// TIA Portal V16 export
// export: Created 2021-11-12T13:31:53.2296923Z, ExportSetting WithDefaults, DisplayName Totally Integrated Automation Portal, DisplayVersion V16 Update 3, DisplayName TIA Portal Version Control Interface, DisplayVersion V16 Update 2, DisplayName TIA Portal Openness, DisplayVersion V16 Update 3, DisplayName SINAMICS Startdrive Advanced, DisplayVersion V16 Update 5, DisplayName SINAMICS Startdrive G130, G150, S120, S150, SINAMICS MV, S210, DisplayVersion V16 Update 5, DisplayName SINAMICS Startdrive G110M, G120, G120C, G120D, G120P, G115D, DisplayVersion V16 Update 5, DisplayName STEP 7 Professional, DisplayVersion V16 Update 3, DisplayName STEP 7 Safety, DisplayVersion V16, DisplayName WinCC UA Professional, DisplayVersion V16 Update 3
DATA_BLOCK "STATUS_000+UH10"   // DB60
{ S7_Optimized_Access := 'TRUE' }
VERSION : 0.1
// stored: AutoNumber true, DBAccessibleFromOPCUA true, IsOnlyStoredInLoadMemory false, IsRetainMemResEnabled false, IsWriteProtectedInAS false, MemoryReserve 100
   VAR
      xxxxx___BinarySensors___xxxxx : Byte;
      xxxxx___BinaryOthers___xxxxx : Byte;
      EC01_3 : Bool;   // Chlazení rozvaděče Vstupní filtr Centrální pult UH10 OK
      FC21_14 : Bool;   // Napájení 230V Centrální pult UH10 UPS OK
      FC22_14 : Bool;   // Napájení 230V Centrální pult UH10 Zásuvky OK
      FB02_14 : Bool;   // Napájení 230V Centrální pult UH10 Servisní zásuvky OK
      SF02_14 : Bool;   // Start automat
      SF03_14 : Bool;   // Nulování poruchy
      SF04_14 : Bool;   // Reset bezpečnostního okruhu
      "I452.7" : Bool;   // Rezerva res10
      SF06_14 : Bool;   // Osvětlení kamer Zóna 1
      SF07_14 : Bool;   // Osvětlení kamer Zóna 2
      SF08_14 : Bool;   // Osvětlení kamer Zóna 3
      SF09_14 : Bool;   // Osvětlení kamer Zóna 4
      "I453.4" : Bool;   // Rezerva res15
      "I453.5" : Bool;   // Rezerva res16
      "I453.7" : Bool;   // Rezerva res4
      SF14_22 : Bool;   // Blokování pásu v peci 1
      SF15_22 : Bool;   // Blokování pásu v peci 2
      SF16_22 : Bool;   // Blokování pásu v peci 3
      SF17_22 : Bool;   // Blokování dopravníku chlazení 1
      SF18_22 : Bool;   // Blokování pásu v peci 4
      SF19_22 : Bool;   // Blokování dopravníku chlazení 2
      SF20_22 : Bool;   // Blokování pásu v peci 5
      SF21_22 : Bool;   // Blokování dopravníku chlazení 3
      SF22_14 : Bool;   // Přemostění Safe move 2R1, 2R2
      "I455.1" : Bool;   // Rezerva res14
      "I455.7" : Bool;   // Rezerva res8
      "I456.1" : Bool;   // Rezerva 2R3
      "I456.2" : Bool;   // Rezerva 2R4
      "I456.3" : Bool;   // Rezerva 2R5
      "I456.4" : Bool;   // Rezerva 2R6
      "I456.5" : Bool;   // Rezerva res14
      "I456.6" : Bool;   // Rezerva res15
      "I456.7" : Bool;   // Rezerva
      xxxxx___InterfaceSignals___xxxxx : Byte;
      SumErr : Bool;   // Sum of significant errors
      PwrOK : Bool;   // Significant switches ON
      xxxxx___AnalogueSensors___xxxxx : Byte;
      xxxxx___Drives___xxxxx : Byte;
      xxxxx___Other___xxxxx : Byte;
      xxxxx__Alarms___xxxxx : Byte;
      EC01_4 : Struct   // Distributor cooling Input filter Central pult UH10 is OK / Chlazení rozvaděče Vstupní filtr Centrální pult UH10 OK
         Main { S7_SetPoint := 'True'} : "UDT_Status_main";
         Specific { S7_SetPoint := 'True'} : "UDT_DI_Mon_Status_specific";
         Error { S7_SetPoint := 'True'} : "UDT_Error01";
      END_STRUCT;
      FC21_15 : Struct   // Power supply 230V Central pult UH10 UPS is OK / Napájení 230V Centrální pult UH10 UPS OK
         Main { S7_SetPoint := 'True'} : "UDT_Status_main";
         Specific { S7_SetPoint := 'True'} : "UDT_DI_Mon_Status_specific";
         Error { S7_SetPoint := 'True'} : "UDT_Error01";
      END_STRUCT;
      FC22_15 : Struct   // Power supply 230V Central pult UH10 Socket is OK / Napájení 230V Centrální pult UH10 Zásuvky OK
         Main { S7_SetPoint := 'True'} : "UDT_Status_main";
         Specific { S7_SetPoint := 'True'} : "UDT_DI_Mon_Status_specific";
         Error { S7_SetPoint := 'True'} : "UDT_Error01";
      END_STRUCT;
      FB02_15 : Struct   // Power supply 230V Central pult UH10 Service socket is OK / Napájení 230V Centrální pult UH10 Servisní zásuvky OK
         Main { S7_SetPoint := 'True'} : "UDT_Status_main";
         Specific { S7_SetPoint := 'True'} : "UDT_DI_Mon_Status_specific";
         Error { S7_SetPoint := 'True'} : "UDT_Error01";
      END_STRUCT;
      SF22_15 : Struct   // By-pass Safe move 2R1, 2R2 / Přemostění Safe move 2R1, 2R2
         Main { S7_SetPoint := 'True'} : "UDT_Status_main";
         Specific { S7_SetPoint := 'True'} : "UDT_DI_Mon_Status_specific";
         Error { S7_SetPoint := 'True'} : "UDT_Error01";
      END_STRUCT;
      ES : Struct   // E-stop
         Main { S7_SetPoint := 'True'} : "UDT_Status_main";
         Specific { S7_SetPoint := 'True'} : "UDT_DI_Mon_Status_specific";
         Error { S7_SetPoint := 'True'} : "UDT_Error01";
      END_STRUCT;
   END_VAR
BEGIN
END_DATA_BLOCK
